# EPICS autosave request: stdApp/Db/userCalcs10_settings.req
# FILE... userCalcs10_settings.req
# USAGE.. userCalcs10.db fields autosave'd.

file swait_settings.req P=$(P)userCalc1
file swait_settings.req P=$(P)userCalc2
file swait_settings.req P=$(P)userCalc3
file swait_settings.req P=$(P)userCalc4
file swait_settings.req P=$(P)userCalc5
file swait_settings.req P=$(P)userCalc6
file swait_settings.req P=$(P)userCalc7
file swait_settings.req P=$(P)userCalc8
file swait_settings.req P=$(P)userCalc9
file swait_settings.req P=$(P)userCalc10
